// TIA Portal V16 export
// export: Created 2023-08-28T09:37:56.54156Z, ExportSetting WithDefaults, DisplayName Totally Integrated Automation Portal, DisplayVersion V16 Update 6, DisplayName TIA Portal Version Control Interface, DisplayVersion V16 Update 2, DisplayName TIA Portal Openness, DisplayVersion V16 Update 6, DisplayName STEP 7 Professional, DisplayVersion V16 Update 6, DisplayName STEP 7 Safety, DisplayVersion V16, DisplayName WinCC Advanced, DisplayVersion V16 Update 6
TYPE "typeDataInverter_Word"
// stored: IsFailsafeCompliant false
   STRUCT
      typeDataInverter_int : Array[0..0] of Int;   // Typ danej Int, falownik
   END_STRUCT;
END_TYPE
